// TIA Portal V16 export
// export: Created 2021-07-12T14:47:15.0520953Z, ExportSetting WithDefaults, DisplayName Totally Integrated Automation Portal, DisplayVersion V16, DisplayName TIA Portal Version Control Interface, DisplayVersion V16, DisplayName TIA Portal Openness, DisplayVersion V16, DisplayName STEP 7 Professional, DisplayVersion V16, DisplayName STEP 7 Safety, DisplayVersion V16, DisplayName WinCC Professional, DisplayVersion V16
DATA_BLOCK "SimaHydTO_HMIConnection"   // DB33100
TITLE = SimaHydTO_HMIConnection
{ S7_Optimized_Access := 'TRUE' }
FAMILY : SimaHydTO
VERSION : 1.0
// Connection data to HMI
// stored: AutoNumber true, DBAccessibleFromOPCUA true, InstanceOfName SimaHydTO_typeHMIConnection, InstanceOfType UDT, IsOnlyStoredInLoadMemory false, IsWriteProtectedInAS false
"SimaHydTO_typeHMIConnection"
   // VAR
   //    AxisData { S7_SetPoint := 'True'} : "SimaHydTO_typeHMIConnectionAxisData";
   //    AxisToData { S7_SetPoint := 'True'} : "SimaHydTO_typeHMIConnectionAxisToData";
   //    AxisSelector { S7_SetPoint := 'True'} : "SimaHydTO_typeHMIConnectionAxisSelector";
   //    BasicAxisControl { S7_SetPoint := 'True'} : "SimaHydTO_typeHMIConnectionBasicAxisControl";
   //    GetCharacteristics { S7_SetPoint := 'True'} : "SimaHydTO_typeHMIConnectionGetCharacteristicInterface";
   //    HmiData { S7_SetPoint := 'True'} : "SimaHydTO_typeHMIConnectionHmiData";
   //    VCharEditor { S7_SetPoint := 'True'} : "SimaHydTO_typeHMIConnectionVCharEditor";
   //    AdvancedAxisControl { S7_SetPoint := 'True'} : "SimaHydTO_typeHMIConnectionAdvancedAxisControl";
   //    ParameterSettings { S7_SetPoint := 'True'} : "SimaHydTO_typeHMIConnectionParameterSettings";
   // END_VAR
BEGIN
   GetCharacteristics.ConfigData.safetyDistance := 100.0;
END_DATA_BLOCK
